TYPE ST_ControlWinch :
STRUCT
	length: LREAL;
	length_t: LREAL;
	length_tt: LREAL;
END_STRUCT
END_TYPE

(* stored: Version 1.1.0.1, ProductVersion 3.1.4022.7
   DUT ST_ControlWinch: Id {2861df26-d324-4aad-9d17-5404fa9cc812} *)
